TYPE U_OdriveUintBytes :
UNION
    Value : UINT;
    Bytes : ARRAY[0..1] OF BYTE;
END_UNION
END_TYPE

(* stored: Version 1.1.0.1
   DUT U_OdriveUintBytes: Id {3DD93AAE-8480-45CF-8CEE-C8E9D3B47EF4} *)
